FUNCTION F_BarToEng : LREAL
VAR_INPUT
	fBar : LREAL;
	
END_VAR
VAR
END_VAR

F_BarToEng := fBar*1E5;

END_FUNCTION

(* stored: Version 1.1.0.1, ProductVersion 3.1.4024.10
   POU F_BarToEng: Id {08df1a0b-1dfe-44e5-a3b6-086d5c827725}, SpecialFunc None *)
